PROGRAM Step_5_Grading //Grading Line
VAR
//--------------------Internals--------------------
	LocalSafety_5  : BOOL;
	
	
	
	
//----------------------Manual Mode---------------------------	
 		JOGGradingVFD2FWD : BOOL; //HMI
		JOGGradingVFD2REV : BOOL;	
	
	
	
// Edge detectors
    rtPullRope_5 : R_TRIG;      // Rising edge Pull Rope	
	
	
	
	
	
	
	
	
	
	
	
	
	
	
	
	
	
	
	
	
END_VAR

//----------------------Safety--------------------

LocalSafety_5  := NOT VFD2Faulted;


//---------------------Defaults-------------------

Step5_RedFlash    := FALSE;
Step5_RedSteady    := FALSE;
Step5_YellowSteady := FALSE;
Step5_YellowFlash := FALSE;
Step5_GreenSteady  := FALSE;
Step5_GreenFlash  := FALSE;
GradingVFD2FWD := FALSE;
GradingVFD2REV := FALSE;

rtPullRope_5(CLK := GradingRopePull);


// Stop button or lost permissive or lost local safety → go to IDLE immediately
IF CycleStopPB OR NOT Permissive OR NOT LocalSafety_5 THEN
    Step5_State := 0; // IDLE
END_IF	



// ----------------------------------- Manual override (when AutoMode = FALSE) ---------------------------------------
IF NOT AutoMode THEN
    GradingVFD2FWD := FALSE;
    GradingVFD2REV := FALSE;

    IF Permissive AND LocalSafety_5 THEN
        // Only run FWD if REV jog is NOT pressed
        IF JOGGradingVFD2FWD AND NOT JOGGradingVFD2REV THEN
            GradingVFD2FWD := TRUE;
        END_IF

        // Only run REV if FWD jog is NOT pressed
        IF JOGGradingVFD2REV AND NOT JOGGradingVFD2FWD THEN
            GradingVFD2REV := TRUE;
        END_IF
    END_IF;

    RETURN;
END_IF



//--------------------------AutoMode---------------------------------------------------------------------------
CASE Step5_State OF

0: // Stopped  


GradingVFD2FWD := FALSE;
GradingVFD2REV := FALSE;

IF CycleStartPB OR rtPullRope_5.Q THEN
    Step5_State := 5; // IDLE
END_IF	


5: // Running/Standby
   

IF NOT GradingEndLimit THEN
   GradingVFD2FWD := TRUE;   // start running
ELSE
	GradingVFD2FWD := FALSE;
END_IF;


IF rtPullRope_5.Q THEN
	Step5_State := 0;

END_IF





END_CASE;

END_PROGRAM

(* stored: Version 1.1.0.1
   POU Step_5_Grading: Id {c380b0e7-991b-4137-87b9-01a5f8095264}, SpecialFunc None *)
